{attribute 'qualified_only'}
VAR_GLOBAL
	nTestValue			: INT;
END_VAR

(* stored: Version 1.1.0.1, ProductVersion 3.1.4024.2
   GVL GVL: Id {209456ab-e551-4b1e-ad66-c6af7911a80e} *)
